// TIA Portal V19 export
FUNCTION_BLOCK "TYPIC_C301_IF_VEN"   // FB5, FBD
TITLE = TYPIC_C301_IF_VEN: Ventilator
{ S7_Optimized_Access := 'TRUE' }
AUTHOR : OCOTECH
FAMILY : Typical
NAME : C301.701
// Logisch Object Besturing: C301.701
// 
// De interne functie ventilator verzorgt de interne besturing, bewaking en fysieke aansturing van een aan/uit ventilator.
// 
// Een langsventilator heeft 2 mogelijke draairichtingen:
//  Rijrichting
//  Tegenrij
// Een ingangsventilator heeft 1 mogelijke draairichting:
//  Rijrichting
// stored: MemoryReserve 10, SetENOAutomatically false
   VAR_INPUT
      PULS_100ms { ExternalAccessible := 'False'; ExternalVisible := 'False'; ExternalWritable := 'False'} : Bool;   // Puls, 1 PLC-cyclus hoog, 1 keer per 100 ms
      PULS_1s { ExternalAccessible := 'False'; ExternalVisible := 'False'; ExternalWritable := 'False'} : Bool;   // Puls, 1 PLC-cyclus hoog, 1 keer per seconde
      EXT_AUT { ExternalAccessible := 'False'; ExternalVisible := 'False'; ExternalWritable := 'False'} : Bool;   // Externe (hoofd) beveiliging (1 = OK)
      EXT_HW { ExternalAccessible := 'False'; ExternalVisible := 'False'; ExternalWritable := 'False'} : Bool;   // Sturings hardware (PLC) bewaking (1 = OK)
      IN_HND { ExternalAccessible := 'False'; ExternalVisible := 'False'; ExternalWritable := 'False'} : Bool;   // Terugmelding aansturing via hand (hardware)
      IN_POS { ExternalAccessible := 'False'; ExternalVisible := 'False'; ExternalWritable := 'False'} : Bool;   // Terugmelding aansturing in rijrichting
      IN_NEG { ExternalAccessible := 'False'; ExternalVisible := 'False'; ExternalWritable := 'False'} : Bool;   // Terugmelding aansturing tegenrijrichting
      IN_AUT { ExternalAccessible := 'False'; ExternalVisible := 'False'; ExternalWritable := 'False'} : Bool;   // Status thermische beveiliging (1 = OK)
      IN_PTC { ExternalAccessible := 'False'; ExternalVisible := 'False'; ExternalWritable := 'False'} : Bool;   // Detectie hoge temperatuur in de motorwikkelingen (1 = OK)
      IN_TRL { ExternalAccessible := 'False'; ExternalVisible := 'False'; ExternalWritable := 'False'} : Word;   // Detectie trillingen (onbalans)
      IN_SCW { ExternalAccessible := 'False'; ExternalVisible := 'False'; ExternalWritable := 'False'} : Bool;   // Werkschakelaar (1 = AAN)
      IN_STO { ExternalAccessible := 'False'; ExternalVisible := 'False'; ExternalWritable := 'False'} : Bool;   // Storingsmelding MCC (1 = OK)
      IN_STS1 { ExternalAccessible := 'False'; ExternalVisible := 'False'; ExternalWritable := 'False'} : Bool;   // Status motorlade in (1 = Ingeschakeld )
      IN_STS2 { ExternalAccessible := 'False'; ExternalVisible := 'False'; ExternalWritable := 'False'} : Bool;   // Status motorlade in test (1 = In Test)
      IN_STS3 { ExternalAccessible := 'False'; ExternalVisible := 'False'; ExternalWritable := 'False'} : Bool;   // Status motorlade uitgereden (1 = Uitgereden)
      IN_STR1 { ExternalAccessible := 'False'; ExternalVisible := 'False'; ExternalWritable := 'False'} : Real;   // Analoge meting ventilator fasestroom 1
      IN_STR2 { ExternalAccessible := 'False'; ExternalVisible := 'False'; ExternalWritable := 'False'} : Real;   // Analoge meting ventilator fasestroom 2
      IN_STR3 { ExternalAccessible := 'False'; ExternalVisible := 'False'; ExternalWritable := 'False'} : Real;   // Analoge meting ventilator fasestroom 3
      CFG_2RI { ExternalAccessible := 'False'; ExternalVisible := 'False'; ExternalWritable := 'False'} : Bool;   // TRUE = Ventilator kan in twee richtingen draaien (i.p.v. enkel een richting)
      CFG_UTYD { ExternalAccessible := 'False'; ExternalVisible := 'False'; ExternalWritable := 'False'} : Time;   // Omschakeltijd, tijd die nodig is om uit te bollen in een richting vooraleer de andere richting gestart mag worden.
      CFG_TYD_FB { ExternalAccessible := 'False'; ExternalVisible := 'False'; ExternalWritable := 'False'} : Time;   // Vertragingstijd storing foute terugmelding
      CFG_TYD_TRL { ExternalAccessible := 'False'; ExternalVisible := 'False'; ExternalWritable := 'False'} : Time;   // Vertragingstijd storing onbalans
      CFG_TRL_MAX { ExternalAccessible := 'False'; ExternalVisible := 'False'; ExternalWritable := 'False'} : Real;   // Hoogste waarde scalering trillingsmeting
      CFG_TRL_MIN { ExternalAccessible := 'False'; ExternalVisible := 'False'; ExternalWritable := 'False'} : Real;   // Laagste waarde scalering trillingsmeting
      CFG_TRL_HOOG { ExternalAccessible := 'False'; ExternalVisible := 'False'; ExternalWritable := 'False'} : Real;   // Schakeldrempel hoog trillingsmeting (onbalans)
   END_VAR
   VAR_OUTPUT
      VAR_IF_VEN { ExternalAccessible := 'False'; ExternalVisible := 'False'; ExternalWritable := 'False'} : "C301_VAR_IF_VEN_TYPIC";   // Struct met alle variabelen naar bovenliggende functies
      OUT_POS { ExternalAccessible := 'False'; ExternalVisible := 'False'; ExternalWritable := 'False'} : Bool;   // Aansturen contactor rijrichting
      OUT_NEG { ExternalAccessible := 'False'; ExternalVisible := 'False'; ExternalWritable := 'False'} : Bool;   // Aansturen contactor tegenrij
      OUT_RES { ExternalAccessible := 'False'; ExternalVisible := 'False'; ExternalWritable := 'False'} : Bool;   // Reset van de motorlade storingen
   END_VAR
   VAR_IN_OUT
      STU_IF_VEN : "C301_STU_IF_VEN_TYPIC";   // Struct met alle sturingen van de subfunctie (SF) calamiteitendoorsteek van 3B
      STU_VGV_VEN_AAN : Bool;   // Vrijgave inschakelen
   END_VAR
   VAR
      STO { ExternalWritable := 'False'} : Struct   // Storingen
         A001 : Bool;   // Beveiliging aangesproken
         A002 : Bool;   // Algemene storing MCC
         A003 : Bool;   // Te hoge temperatuur in de wikkelingen van de motor van de ventilator
         A004 : Bool;   // De ventilator is in onbalans
         A005 : Bool;   // Fout stroommeting fase 1
         A006 : Bool;   // Fout stroommeting fase 2
         A007 : Bool;   // Fout stroommeting fase 3
         A008 : Bool;   // Motorlade uitgeschakeld
         A009 : Bool;   // Motorlade in test
         A010 : Bool;   // Motorlade uitgereden
         A011 : Bool;   // Draadbreuk trillingsmeting
         A012 : Bool;   // Meetbereik trillingsmeting overschreden
         AT01 : Bool;   // Discordantie motor: terugmelding niet ontvangen
         AT02 : Bool;   // Discordantie motor: terugmelding blijft aanwezig
         AT03 : Bool;   // Discordantie motor: terugmeldingen Positief en negatief tegelijkertijd
         M001 : Bool;   // Werkschakelaar uitgeschakeld
      END_STRUCT;
      VAR { ExternalWritable := 'False'} : Struct   // Variabelen
         STS_AAN { ExternalAccessible := 'False'; ExternalVisible := 'False'} : Bool;   // TRUE = Ventilator is aangestuurd FALSE = Uit
         DIR_POS { ExternalAccessible := 'False'; ExternalVisible := 'False'} : Bool;   // TRUE = Ventilator draait in positieve richting (rijrichting)
         DIR_NEG { ExternalAccessible := 'False'; ExternalVisible := 'False'} : Bool;   // TRUE = Ventilator draait in negatieve richting (tegenrij)
         BMO_HAND { ExternalAccessible := 'False'; ExternalVisible := 'False'} : Bool;   // TRUE = Ventilator in hand geschakeld FALSE = niet in hand
         TYD_TOT_AAN { ExternalAccessible := 'False'; ExternalVisible := 'False'} : LInt;   // Totaal aantal draaiuren
         TYD_TOT_AAN_UUR { ExternalAccessible := 'False'; ExternalVisible := 'False'} : LInt;   // Totaal aantal draaiuren
         ENE_MWA1 { ExternalAccessible := 'False'; ExternalVisible := 'False'} : Real;   // Stroommeting fase 1
         ENE_MWA2 { ExternalAccessible := 'False'; ExternalVisible := 'False'} : Real;   // Stroommeting fase 2
         ENE_MWA3 { ExternalAccessible := 'False'; ExternalVisible := 'False'} : Real;   // Stroommeting fase 3
         TRL_MWA { ExternalAccessible := 'False'; ExternalVisible := 'False'} : Real;   // Trillingsmeting
         EXT_AUT { ExternalAccessible := 'False'; ExternalVisible := 'False'} : Bool;   // Externe (hoofd) beveiliging aangesproken
         EXT_HW { ExternalAccessible := 'False'; ExternalVisible := 'False'} : Bool;   // Sturings hardware (PLC) in storing
      END_STRUCT;
   END_VAR
BEGIN

REGION Network 1: START
END_REGION

REGION Network 2: +++ Metingen +++
   // Inlezen van de 3 stroommetingen van iedere fase van de motor en inlezen van de trillingsmeting.
END_REGION

REGION Network 3: +++ Storingen +++
   // Verwerken van de storingsmeldingen (inputs).
END_REGION

REGION Network 4: Storing A001: Beveiliging aangesproken
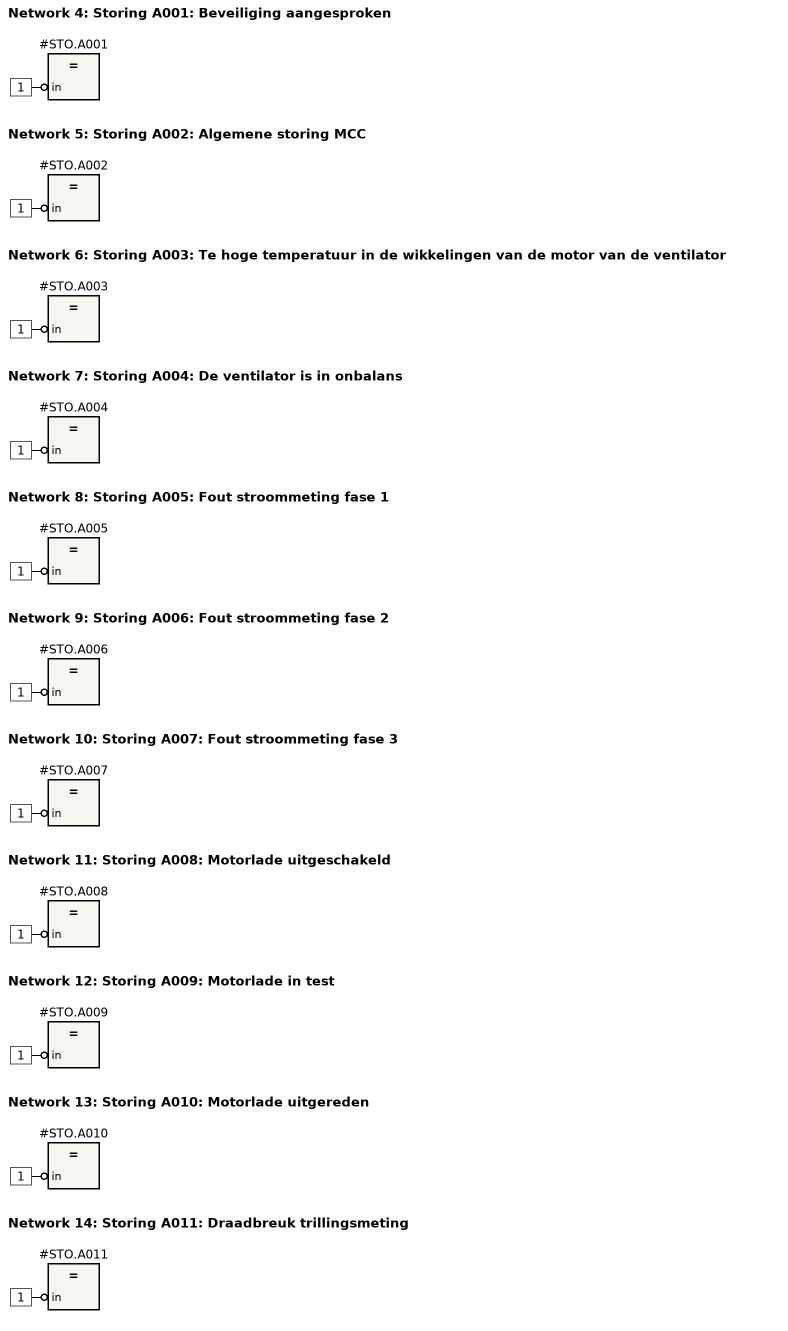
   #STO.A001 := NOT 1;
END_REGION

REGION Network 5: Storing A002: Algemene storing MCC
   #STO.A002 := NOT 1;
END_REGION

REGION Network 6: Storing A003: Te hoge temperatuur in de wikkelingen van de motor van de ventilator
   #STO.A003 := NOT 1;
END_REGION

REGION Network 7: Storing A004: De ventilator is in onbalans
   #STO.A004 := NOT 1;
END_REGION

REGION Network 8: Storing A005: Fout stroommeting fase 1
   #STO.A005 := NOT 1;
END_REGION

REGION Network 9: Storing A006: Fout stroommeting fase 2
   #STO.A006 := NOT 1;
END_REGION

REGION Network 10: Storing A007: Fout stroommeting fase 3
   #STO.A007 := NOT 1;
END_REGION

REGION Network 11: Storing A008: Motorlade uitgeschakeld
   #STO.A008 := NOT 1;
END_REGION

REGION Network 12: Storing A009: Motorlade in test
   #STO.A009 := NOT 1;
END_REGION

REGION Network 13: Storing A010: Motorlade uitgereden
   #STO.A010 := NOT 1;
END_REGION

REGION Network 14: Storing A011: Draadbreuk trillingsmeting
   #STO.A011 := NOT 1;
END_REGION

REGION Network 15: Storing A012: Meetbereik trillingsmeting overschreden
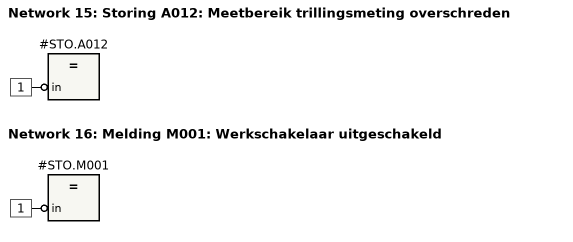
   #STO.A012 := NOT 1;
END_REGION

REGION Network 16: Melding M001: Werkschakelaar uitgeschakeld
   #STO.M001 := NOT 1;
END_REGION

REGION Network 17: +++ Motorsturing +++
   // Aansturen en bewaking van de motor.
END_REGION

REGION Network 18: +++ Urentellers +++
   // Tellen van de tijdsduur dat motor draait of stilstaat.
END_REGION

REGION Network 19 (SCL): EINDE
   // Variabelen van intern scada rakvlak naar outputs copieren
   #VAR_IF_VEN.STS_AAN := #VAR.STS_AAN;
   #VAR_IF_VEN.DIR_POS := #VAR.DIR_POS;
   #VAR_IF_VEN.DIR_NEG := #VAR.DIR_NEG;
   #VAR_IF_VEN.BMO_HAND := #VAR.BMO_HAND;
   #VAR_IF_VEN.TYD_TOT_AAN := #VAR.TYD_TOT_AAN;
   #VAR_IF_VEN.TYD_TOT_AAN_UUR := #VAR.TYD_TOT_AAN_UUR;
   #VAR_IF_VEN.ENE_MWA1 := #VAR.ENE_MWA1;
   #VAR_IF_VEN.ENE_MWA2 := #VAR.ENE_MWA2;
   #VAR_IF_VEN.ENE_MWA3 := #VAR.ENE_MWA3;
   #VAR_IF_VEN.TRL_MWA := #VAR.TRL_MWA;
   #VAR_IF_VEN.EXT_AUT := #VAR.EXT_AUT;
   #VAR_IF_VEN.EXT_HW := #VAR.EXT_HW;
   #VAR_IF_VEN.STO := #STO;
END_REGION
END_FUNCTION_BLOCK
